FUNCTION TryConvert_TIME_TO_UDINT : BOOL
VAR_INPUT
	in : TIME;
	out : REFERENCE TO UDINT;
END_VAR

out := TIME_TO_UDINT(in);
TryConvert_TIME_TO_UDINT := TRUE;

END_FUNCTION

(* stored: Version 1.1.0.1, ProductVersion 3.1.4024.12
   POU TryConvert_TIME_TO_UDINT: Id {2b72bf8b-a737-492b-bdb9-889bb77500a6}, SpecialFunc None *)
